// TIA Portal V17 export
// export: Created 2023-02-23T17:16:27.2939153Z, ExportSetting WithDefaults, DisplayName Totally Integrated Automation Portal, DisplayVersion V17, DisplayName TIA Portal Openness, DisplayVersion V17, DisplayName TIA Portal Version Control Interface, DisplayVersion V17, DisplayName TIA Portal Test Suite Advanced, DisplayVersion V17, DisplayName STEP 7 Professional, DisplayVersion V17, DisplayName SIMATIC Energy Suite, DisplayVersion V17, DisplayName STEP 7 Safety, DisplayVersion V17, DisplayName WinCC Professional, DisplayVersion V17
FUNCTION_BLOCK "MAN_ControlLine"   // FB2, LAD
TITLE = Control Line - Sequential algorithm
{ S7_Optimized_Access := 'TRUE' }
VERSION : 0.1
// stored: AutoNumber true, IsIECCheckEnabled false, IsRetainMemResEnabled false, MemoryReserve 100, SetENOAutomatically false, UDAEnableTagReadback false
   VAR_INPUT
      ButtonStart : Bool;
      ButtonStop : Bool;
      ModeManual : Bool;
      ModeAuto : Bool;
      GlobalError : Bool;
      FirstScan : Bool;
   END_VAR
   VAR_OUTPUT
      StartLine : Bool;
      StopLine : Bool;
      AlarmSiren : Bool;
   END_VAR
   VAR
      s1 : Bool;
      s2 : Bool;
      s3 : Bool;
      s4 : Bool;
      P_ButtonStart_1 : Bool;
      P_ButtonStart_2 : Bool;
      IEC_Timer_0_Instance { ExternalAccessible := 'False'; ExternalVisible := 'False'; ExternalWritable := 'False'} : TP_TIME;
      Run { S7_SetPoint := 'True'} : Bool;
      N_Run : Bool;
   END_VAR
   VAR_TEMP   // added for the SCL form of the ladder/FBD networks
      _w1 : Bool;
   END_VAR
BEGIN

REGION Network 1: Step 2-1
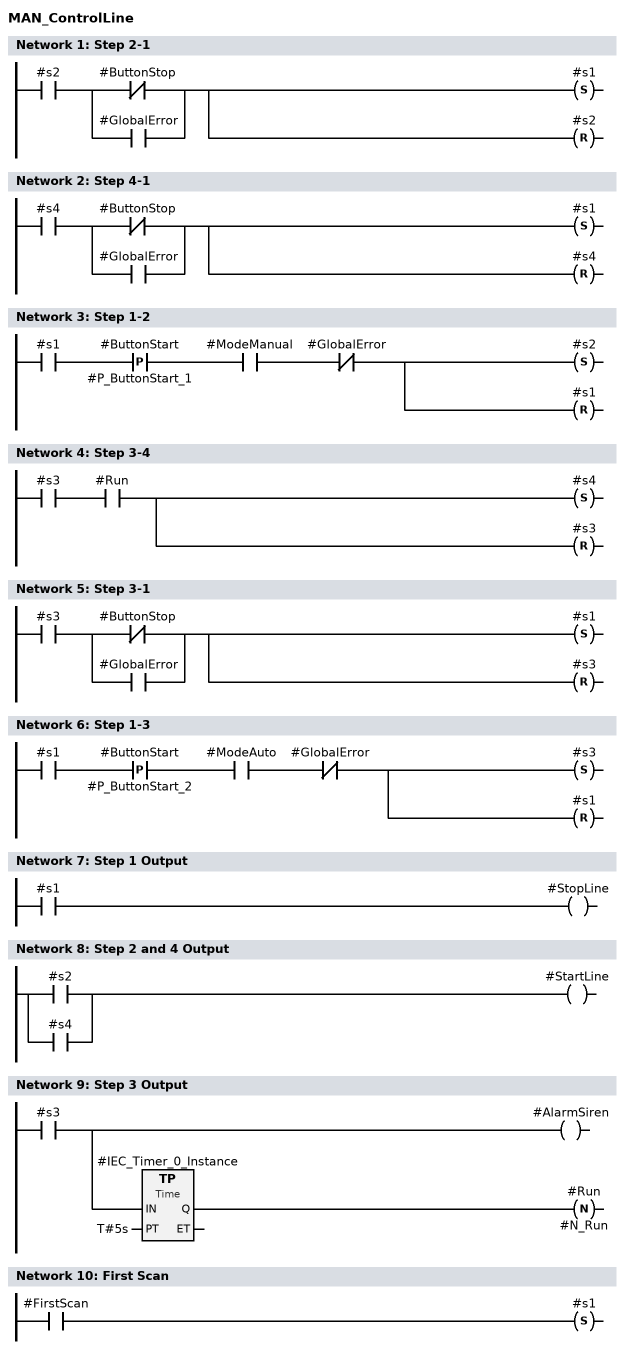
   RUNG wire#powerrail
      Contact( #s2 )
      wire#w1
      I_Contact( #ButtonStop )
      wire#w2
      S_Coil( #s1 )
   END_RUNG
   RUNG wire#w1
      Contact( #GlobalError )
   END_RUNG wire#w2
   RUNG wire#w2
      R_Coil( #s2 )
   END_RUNG
   // the same network as SCL:
   IF #s2 AND (NOT #ButtonStop OR #GlobalError) THEN
       #s1 := TRUE;
       #s2 := FALSE;
   END_IF;
END_REGION

REGION Network 2: Step 4-1
   RUNG wire#powerrail
      Contact( #s4 )
      wire#w1
      I_Contact( #ButtonStop )
      wire#w2
      S_Coil( #s1 )
   END_RUNG
   RUNG wire#w1
      Contact( #GlobalError )
   END_RUNG wire#w2
   RUNG wire#w2
      R_Coil( #s4 )
   END_RUNG
   // the same network as SCL:
   IF #s4 AND (NOT #ButtonStop OR #GlobalError) THEN
       #s1 := TRUE;
       #s4 := FALSE;
   END_IF;
END_REGION

REGION Network 3: Step 1-2
   RUNG wire#powerrail
      Contact( #s1 )
      P_Contact(operand := #ButtonStart, bit := #P_ButtonStart_1)
      Contact( #ModeManual )
      I_Contact( #GlobalError )
      wire#w1
      S_Coil( #s2 )
   END_RUNG
   RUNG wire#w1
      R_Coil( #s1 )
   END_RUNG
   // the same network as SCL:
   #_w1 := #s1 AND #ButtonStart AND NOT #P_ButtonStart_1;   // rising edge of #ButtonStart
   #P_ButtonStart_1 := #ButtonStart;
   IF #_w1 AND #ModeManual AND NOT #GlobalError THEN
       #s2 := TRUE;
       #s1 := FALSE;
   END_IF;
END_REGION

REGION Network 4: Step 3-4
   RUNG wire#powerrail
      Contact( #s3 )
      Contact( #Run )
      wire#w1
      S_Coil( #s4 )
   END_RUNG
   RUNG wire#w1
      R_Coil( #s3 )
   END_RUNG
   // the same network as SCL:
   IF #s3 AND #Run THEN
       #s4 := TRUE;
       #s3 := FALSE;
   END_IF;
END_REGION

REGION Network 5: Step 3-1
   RUNG wire#powerrail
      Contact( #s3 )
      wire#w1
      I_Contact( #ButtonStop )
      wire#w2
      S_Coil( #s1 )
   END_RUNG
   RUNG wire#w1
      Contact( #GlobalError )
   END_RUNG wire#w2
   RUNG wire#w2
      R_Coil( #s3 )
   END_RUNG
   // the same network as SCL:
   IF #s3 AND (NOT #ButtonStop OR #GlobalError) THEN
       #s1 := TRUE;
       #s3 := FALSE;
   END_IF;
END_REGION

REGION Network 6: Step 1-3
   RUNG wire#powerrail
      Contact( #s1 )
      P_Contact(operand := #ButtonStart, bit := #P_ButtonStart_2)
      Contact( #ModeAuto )
      I_Contact( #GlobalError )
      wire#w1
      S_Coil( #s3 )
   END_RUNG
   RUNG wire#w1
      R_Coil( #s1 )
   END_RUNG
   // the same network as SCL:
   #_w1 := #s1 AND #ButtonStart AND NOT #P_ButtonStart_2;   // rising edge of #ButtonStart
   #P_ButtonStart_2 := #ButtonStart;
   IF #_w1 AND #ModeAuto AND NOT #GlobalError THEN
       #s3 := TRUE;
       #s1 := FALSE;
   END_IF;
END_REGION

REGION Network 7: Step 1 Output
   RUNG wire#powerrail
      Contact( #s1 )
      Coil( #StopLine )
   END_RUNG
   // the same network as SCL:
   #StopLine := #s1;
END_REGION

REGION Network 8: Step 2 and 4 Output
   RUNG wire#powerrail
      Contact( #s2 )
      wire#w1
      Coil( #StartLine )
   END_RUNG
   RUNG wire#powerrail
      Contact( #s4 )
   END_RUNG wire#w1
   // the same network as SCL:
   #StartLine := #s2 OR #s4;
END_REGION

REGION Network 9: Step 3 Output
   #AlarmSiren := #s3;
   #IEC_Timer_0_Instance(IN := #s3, PT := T#5s);   // TP
   #Run := NOT #IEC_Timer_0_Instance.Q AND #N_Run;   // falling edge
   #N_Run := #IEC_Timer_0_Instance.Q;
END_REGION

REGION Network 10: First Scan
   RUNG wire#powerrail
      Contact( #FirstScan )
      S_Coil( #s1 )
   END_RUNG
   // the same network as SCL:
   IF #FirstScan THEN #s1 := TRUE; END_IF;
END_REGION
END_FUNCTION_BLOCK
